FUNCTION_BLOCK ZONE_MDLL (* HVAC Zone Model with Local Comms *)
  (* Standard: 61499-1; Classification: Simulation; ApplicationDomain: HVAC; Function: Zone Model *)
  (* Version 0.0, 2006-04-13, JHC, Holobloc Inc *)
  (* Compiler header: package fb.rt.hvac; import fb.rt.net.*; *)
  (* Compiler Java Sun JDK 1.5.0 *)
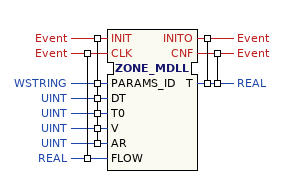
  EVENT_INPUT
    INIT WITH T0, V, AR, DT, PARAMS_ID; (* Initialization Request *)
    CLK WITH FLOW; (* Simulation Clock *)
  END_EVENT
  EVENT_OUTPUT
    INITO WITH T; (* INIT completed *)
    CNF WITH T; (* Simulation step completed *)
  END_EVENT
  VAR_INPUT
    PARAMS_ID : WSTRING := "PARAMS"; (* STEMP, XTEMP, LOAD subscriber channel ID *)
    DT : UINT := 10; (* Clock period, sec *)
    T0 : UINT := 70; (* Initial Temperature, deg F *)
    V : UINT := 5000; (* Zone volume, cu ft *)
    AR : UINT := 20; (* Wall A/R, BTU/hr/deg F *)
    FLOW : REAL; (* Air Flow, CFM *)
  END_VAR
  VAR_OUTPUT
    T : REAL; (* Zone Temperature, deg F *)
  END_VAR
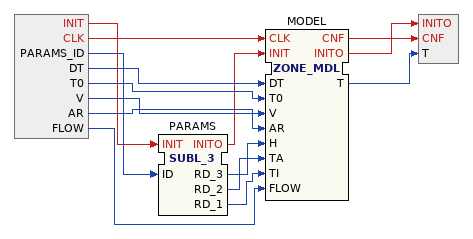
  FBS
    MODEL : ZONE_MDL;
    PARAMS : SUBL_3;
  END_FBS
  EVENT_CONNECTIONS
    MODEL.CNF TO CNF;
    CLK TO MODEL.CLK;
    INIT TO PARAMS.INIT;
    PARAMS.INITO TO MODEL.INIT;
    MODEL.INITO TO INITO;
  END_CONNECTIONS
  DATA_CONNECTIONS
    DT TO MODEL.DT;
    T0 TO MODEL.T0;
    V TO MODEL.V;
    AR TO MODEL.AR;
    MODEL.T TO T;
    PARAMS_ID TO PARAMS.ID;
    PARAMS.RD_3 TO MODEL.H;
    PARAMS.RD_2 TO MODEL.TA;
    PARAMS.RD_1 TO MODEL.TI;
    FLOW TO MODEL.FLOW;
  END_CONNECTIONS
END_FUNCTION_BLOCK
